PROGRAM MAIN
VAR
END_VAR

END_PROGRAM

(* stored: Version 1.1.0.1
   POU MAIN: Id {5a6e8b50-8dd8-4eba-9459-28fa6c7e6d6e} *)
